KUKA KRL data list: UTILS.dat

&ACCESS RVO1
&REL 5
DEFDAT UTILS PUBLIC
   GLOBAL ENUM NORMAL_AXIS_T NORMAL_X, NORMAL_Y, NORMAL_Z
   GLOBAL ENUM PROJ_MODE_T PROJ_KEEP_POINT_ROT, PROJ_KEEP_PLANE_ROT
ENDDAT
